TYPE T_CodeBRAND : STRING[9];
END_TYPE

(* stored: Version 1.1.0.1
   DUT T_CodeBRAND: Id {0f6a90b5-e3f1-4b19-8f33-cb1038a41999} *)
